FUNCTION_BLOCK Led
  (* Standard: 61499-2 *)
  (* Version 0.1, 2017-00-16, hpea485, UOA *)
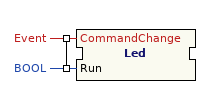
  EVENT_INPUT
    CommandChange WITH Run;
  END_EVENT
  VAR_INPUT
    Run : BOOL;
  END_VAR
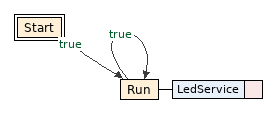
  EC_STATES
    Start;
    Run : LedService;
  END_STATES
  EC_TRANSITIONS
    Start TO Run := true;
    Run TO Run := true;
  END_TRANSITIONS
  ALGORITHM LedService IN C:
if(me->inputEvents.event.CommandChange) {
	LED = me->Run;
}
  END_ALGORITHM
END_FUNCTION_BLOCK
